Staubli VAL3: onEnterEvent.pgx

program onEnterEvent(bool& x_bSave[])
  local bool l_bOk
begin
  pub:libLoad("Disk://page/page_trajectory")
  call pub:main()
end
